TYPE typ_MotionPhasing :
STRUCT
	MC_HaltPhasing				: MC_HaltPhasing;
	MC_PhasingAbsolute			: MC_PhasingAbsolute;
	MC_PhasingRelative			: MC_PhasingRelative;
END_STRUCT
END_TYPE

(* stored: Version 1.1.0.1, ProductVersion 3.1.4022.17
   DUT typ_MotionPhasing: Id {22352df5-192e-459b-9b5c-2f6907cb8760} *)
